// TIA Portal V20 export
TYPE "HMI_Aggr16"
   STRUCT
      OnMan : Bool := FALSE;   // 1=On: On Command in Manual Mode
      OffMan : Bool := TRUE;   // 1=Off: Off Command in Manual Mode
      AutModOp : Bool := FALSE;   // 1=Auto Mode: Auto Mode by Operator
      ManModOp : Bool := TRUE;   // 1=Manual Mode: Manual Mode by Operator
      OosOp : Bool := FALSE;   // 1=Oos Mode: Oos Mode by Operator
      ExtNoOp : Bool := 0;   // Ext Mode for Number of Units: Ext Mode by Operator
      IntNoOp : Bool := 1;   // Int Mode for Number of Units: Int Mode by Operator
      UnitReqOp : USInt := 1;   // Number of Units required from Operator
      ExtSwOp : Bool := 0;   // Ext Mode for Switch: Ext Mode by Operator
      IntSwOp : Bool := 1;   // Int Mode for Switch: Int Mode by Operator
      TimeSwOp : Bool := 0;   // Time Mode for Switch: Time Mode by Operator
      UnitMstrOp : USInt := 1;   // Master Unit from Operator
      ChangeTime : Int := 168;   // Time for Change the Master Agg.[h]
      DelayOn : Real := 0.0;   // Delay Time on [s]
      DelayOff : Real := 0.0;   // Delay Time off [s]
      MaxAggr : USInt := 0;   // max. Number of units
      RunTi01 : DWord := 0;   // Runtime unit 1
      RunTi02 : DWord := 0;   // Runtime unit 2
      RunTi03 : DWord := 0;   // Runtime unit 3
      RunTi04 : DWord := 0;   // Runtime unit 4
      RunTi05 : DWord := 0;   // Runtime unit 5
      RunTi06 : DWord := 0;   // Runtime unit 6
      RunTi07 : DWord := 0;   // Runtime unit 7
      RunTi08 : DWord := 0;   // Runtime unit 8
      RunTi09 : DWord := 0;   // Runtime unit 9
      RunTi10 : DWord := 0;   // Runtime unit 10
      RunTi11 : DWord := 0;   // Runtime unit 11
      RunTi12 : DWord := 0;   // Runtime unit 12
      RunTi13 : DWord := 0;   // Runtime unit 13
      RunTi14 : DWord := 0;   // Runtime unit 14
      RunTi15 : DWord := 0;   // Runtime unit 15
      RunTi16 : DWord := 0;   // Runtime unit 16
      Prio01 : USInt := 1;   // Priority (1 - 99) unit 1
      Prio02 : USInt := 1;   // Priority (1 - 99) unit 2
      Prio03 : USInt := 1;   // Priority (1 - 99) unit 3
      Prio04 : USInt := 1;   // Priority (1 - 99) unit 4
      Prio05 : USInt := 1;   // Priority (1 - 99) unit 5
      Prio06 : USInt := 1;   // Priority (1 - 99) unit 6
      Prio07 : USInt := 1;   // Priority (1 - 99) unit 7
      Prio08 : USInt := 1;   // Priority (1 - 99) unit 8
      Prio09 : USInt := 1;   // Priority (1 - 99) unit 9
      Prio10 : USInt := 1;   // Priority (1 - 99) unit 10
      Prio11 : USInt := 1;   // Priority (1 - 99) unit 11
      Prio12 : USInt := 1;   // Priority (1 - 99) unit 12
      Prio13 : USInt := 1;   // Priority (1 - 99) unit 13
      Prio14 : USInt := 1;   // Priority (1 - 99) unit 14
      Prio15 : USInt := 1;   // Priority (1 - 99) unit 15
      Prio16 : USInt := 1;   // Priority (1 - 99) unit 16
      On { ExternalWritable := 'False'} : Bool;   // 1= Aggr on
      Off { ExternalWritable := 'False'} : Bool := true;   // 1= Aggr off
      PrioOut01 { ExternalWritable := 'False'} : USInt := 1;   // Priority (1 - 99) unit 1
      PrioOut02 { ExternalWritable := 'False'} : USInt := 1;   // Priority (1 - 99) unit 2
      PrioOut03 { ExternalWritable := 'False'} : USInt := 1;   // Priority (1 - 99) unit 3
      PrioOut04 { ExternalWritable := 'False'} : USInt := 1;   // Priority (1 - 99) unit 4
      PrioOut05 { ExternalWritable := 'False'} : USInt := 1;   // Priority (1 - 99) unit 5
      PrioOut06 { ExternalWritable := 'False'} : USInt := 1;   // Priority (1 - 99) unit 6
      PrioOut07 { ExternalWritable := 'False'} : USInt := 1;   // Priority (1 - 99) unit 7
      PrioOut08 { ExternalWritable := 'False'} : USInt := 1;   // Priority (1 - 99) unit 8
      PrioOut09 { ExternalWritable := 'False'} : USInt := 1;   // Priority (1 - 99) unit 9
      PrioOut10 { ExternalWritable := 'False'} : USInt := 1;   // Priority (1 - 99) unit 10
      PrioOut11 { ExternalWritable := 'False'} : USInt := 1;   // Priority (1 - 99) unit 11
      PrioOut12 { ExternalWritable := 'False'} : USInt := 1;   // Priority (1 - 99) unit 12
      PrioOut13 { ExternalWritable := 'False'} : USInt := 1;   // Priority (1 - 99) unit 13
      PrioOut14 { ExternalWritable := 'False'} : USInt := 1;   // Priority (1 - 99) unit 14
      PrioOut15 { ExternalWritable := 'False'} : USInt := 1;   // Priority (1 - 99) unit 15
      PrioOut16 { ExternalWritable := 'False'} : USInt := 1;   // Priority (1 - 99) unit 16
      Start01 { ExternalWritable := 'False'} : Bool;   // 1=Start unit 1
      Start02 { ExternalWritable := 'False'} : Bool;   // 1=Start unit 2
      Start03 { ExternalWritable := 'False'} : Bool;   // 1=Start unit 3
      Start04 { ExternalWritable := 'False'} : Bool;   // 1=Start unit 4
      Start05 { ExternalWritable := 'False'} : Bool;   // 1=Start unit 5
      Start06 { ExternalWritable := 'False'} : Bool;   // 1=Start unit 6
      Start07 { ExternalWritable := 'False'} : Bool;   // 1=Start unit 7
      Start08 { ExternalWritable := 'False'} : Bool;   // 1=Start unit 8
      Start09 { ExternalWritable := 'False'} : Bool;   // 1=Start unit 9
      Start10 { ExternalWritable := 'False'} : Bool;   // 1=Start unit 10
      Start11 { ExternalWritable := 'False'} : Bool;   // 1=Start unit 11
      Start12 { ExternalWritable := 'False'} : Bool;   // 1=Start unit 12
      Start13 { ExternalWritable := 'False'} : Bool;   // 1=Start unit 13
      Start14 { ExternalWritable := 'False'} : Bool;   // 1=Start unit 14
      Start15 { ExternalWritable := 'False'} : Bool;   // 1=Start unit 15
      Start16 { ExternalWritable := 'False'} : Bool;   // 1=Start unit 16
      UnitOn { ExternalWritable := 'False'} : Word := 0;   // Units on Display
      UnitAvail { ExternalWritable := 'False'} : Word := 0;   // Units available Display
      UnitReq { ExternalWritable := 'False'} : USInt := 0;   // Number of Units required
      NoUnitRun { ExternalWritable := 'False'} : USInt := 0;   // Compared Number of Units required/on
      NoUnitAvail { ExternalWritable := 'False'} : USInt := 0;   // Number of Units on and available
      UnitMstr { ExternalWritable := 'False'} : USInt := 0;   // Master Unit
      UnitMissing { ExternalWritable := 'False'} : USInt := 0;   // Units missing
      UnitReserved { ExternalWritable := 'False'} : USInt := 0;   // Reserved Units
      ChangeTime_Out { ExternalWritable := 'False'} : Time := T#0MS;   // Residual Time for Changing Master
      OS_PermOut { ExternalWritable := 'False'} : DWord := 16#FFFF_FFFF;   // Operator Permission: Output for OS
      OS_PermLog { ExternalWritable := 'False'} : DWord := 16#FFFF_FFFF;   // Operator Permission: Output for OS
      OpSt_Out { ExternalWritable := 'False'} : DWord;   // Enabled operator stations
      Status1 { ExternalWritable := 'False'} : DWord;   // Status word 1
      Status2 { ExternalWritable := 'False'} : DWord;   // Status word 2
      AlarmState { ExternalWritable := 'False'} : Word;   // Alarm State for group display / Alarm Status for group display
   END_STRUCT;
END_TYPE
